TYPE ST_SegmentNumberIn :
STRUCT
END_STRUCT
END_TYPE

(* stored: Version 1.1.0.1
   DUT ST_SegmentNumberIn: Id {9faf9233-4bb3-08a6-31bc-2828a927700c} *)
